Staubli VAL3: addStrArray.pgx

public program addStrArray(string& x_sStrIn[], num x_nNum, bool& x_bRes)
  local num l_i
begin
  //建立指定数目的字符串数组
  //x_sStrIn:返回的新数组
  //x_nNum:数组个数
  //x_bRes:函数返回值
  x_bRes=false
  if x_nNum<1
    popUpMsg("新增点个数小于1")
    return
  endIf
  //取整
  x_nNum=roundDown(x_nNum)
  //删除原有的数组
  while size(x_sStrIn)>1
    delete(x_sStrIn[0])
  endWhile
  x_sStrIn[0]=""
  //插入新数据
  for l_i=1 to x_nNum-1
    insert(x_sStrIn[l_i])
  endFor
  x_bRes=true
end
